// TIA Portal V18 export
TYPE "UDT_Store_Scheduler"
// stored: IsFailsafeCompliant false
   STRUCT
      cOpModeNowByScheduler : Byte;
      Monday : Struct
         Comfort { S7_SetPoint := 'True'} : "UDT_DailyScheduler";
         PreComfort { S7_SetPoint := 'True'} : "UDT_DailyScheduler";
      END_STRUCT;
      WorkingDays : Struct
         Comfort { S7_SetPoint := 'True'} : "UDT_DailyScheduler";
         PreComfort { S7_SetPoint := 'True'} : "UDT_DailyScheduler";
      END_STRUCT;
      Saturday : Struct
         Comfort { S7_SetPoint := 'True'} : "UDT_DailyScheduler";
         PreComfort { S7_SetPoint := 'True'} : "UDT_DailyScheduler";
      END_STRUCT;
      Sunday : Struct
         Comfort { S7_SetPoint := 'True'} : "UDT_DailyScheduler";
         PreComfort { S7_SetPoint := 'True'} : "UDT_DailyScheduler";
      END_STRUCT;
      Holiday : Struct
         Comfort { S7_SetPoint := 'True'} : "UDT_DailyScheduler";
         PreComfort { S7_SetPoint := 'True'} : "UDT_DailyScheduler";
      END_STRUCT;
   END_STRUCT;
END_TYPE
